PROGRAM SAFETY
VAR
END_VAR

END_PROGRAM

(* stored: Version 1.1.0.1, ProductVersion 3.1.4024.15
   POU SAFETY: Id {35ba0ba9-0a5d-4f9c-a367-e8f271d5d193}, SpecialFunc None *)
